TYPE CmpConvDivert :	//Version 02 - 06/17/2022
STRUCT
	
	Framework: Framework;
	PuckReady: BOOL;
	Puck: PuckData;
	UnknownPuck: BOOL;
	MainHeartbeatOK: BOOL;
	MainConvRunning: BOOL;
	MainInAuto: BOOL;
	MainBufferFull: BOOL;
	PuckReleaseMain: BOOL;
	PuckReleaseSpur: BOOL;
	StatusInCycleAuto: BOOL;
	FreeRunCycleStop: BOOL;
	senMainBufferFullOff: BOOL;
	senSpurBufferFullOff: BOOL;
	senMainPuckPresentOff: BOOL;
	senMainPuckPresentOn: BOOL;
	
	SpurHeartbeatOK: BOOL;
	SpurConvRunning: BOOL;
	SpurInAuto: BOOL;
	SpurBufferFull: BOOL;
	SpurEmptyRequest: BOOL;
	SpurPurgeMode: BOOL;
	Config: CmpConvDivertConfig;

END_STRUCT
END_TYPE

(* stored: Version 1.1.0.1, ProductVersion 3.1.4024.6
   DUT CmpConvDivert: Id {63d590b6-97ce-4d74-9feb-3aa30b7175ce} *)
